# B&R Automation Studio project Parker_BMM_ST_V5_3147_V12 (part 29)

#### multsave.c
```c
/*************************************************************************************
 * COPYRIGHT --  B&R China
 *************************************************************************************
 * Program: multsave
 * File: multsave.c
 * Author: lijianjun
 * Created: March 06, 2013
 **************************************************************************************
 * Implementation of program multsave --- mold data save/load
 *************************************************************************************/

#include <bur/plctypes.h>
#include <string.h>

#ifdef _DEFAULT_INCLUDES
	#include <AsDefault.h>
#endif

#include "recipe.h"

/**************************************************************************************
** 					 	           macro define								                   **
**************************************************************************************/
#define	S$PVNAME_LENGTH		(C_PVNAME_LENGTH +1)
#define	S$LINE_NUMBER		   (C_LINE_NUMBER   +1)

#define S$WAIT_COMMAND			   10

#define S$ROOT_DISK_SAVE		   100
#define S$ROOT_DISK_LOAD		   200
#define S$ROOT_DISK_CLEAR		   500

#define S$USB_SINGLE_OPEN_SAVE	1000
#define S$USB_SINGLE_CREATE		1100
#define S$USB_SINGLE_WRITE_MEM	1200
#define S$USB_SINGLE_WRITE		   1300

#define S$USB_SINGLE_OPEN_LOAD	2000
#define S$USB_SINGLE_READ_MEM	   2100
#define S$USB_SINGLE_READ			2200

#define S$USB_SINGLE_CLOSE		   3000

#define S$USB_ALL_OPEN_SAVE	   11000
#define S$USB_ALL_CREATE		   11100
#define S$USB_ALL_MEM_ALLOC	   11200
#define S$USB_ALL_MEM_GET	      11300
#define S$USB_ALL_WRITE		      11400
#define S$USB_ALL_MEM_FREE		   11500

#define S$USB_ALL_OPEN_LOAD	   12000
#define S$USB_ALL_ALLOC_MEM	   12100
#define S$USB_ALL_READ			   12200
#define S$USB_ALL_READ_WRITE	   12300
#define S$USB_ALL_FREE_MEM  	   12400

#define S$USB_ALL_CLOSE		      13000

#define S$ERROR_STEP			      40000
/**************************************************************************************
**                            Function Declarations								     **
**************************************************************************************/
void fun_pv_name ();
void fun_pv_info ();
void fun_pv_save (unsigned short index);
void fun_pv_read (unsigned short index);
void fun_pv_clear(unsigned short index);

/**************************************************************************************
****	        		I N I T U P  O F   T H E   T A S K 		 				   ****
**************************************************************************************/
void _INIT _init(void)
{
	memset(pvList,0,sizeof(pvList));
	strcpy(pv_get.modname,"var_mold");

   strcpy(fileSingleName, "mold.usb");		/* file name */
   strcpy(fileAllName, "moldAll.usb");		/* file name */

   strcpy(DataObjOperate.ModName,"recMold");
   strcpy(DataObjOperate.Status,"");
   DataObjOperate.InitStep = 100;

   gUserPara.VarNew = 0;
}  /* end of _INIT */

/**************************************************************************************
****				C Y C L I C   P A R T   O F   T H E   T A S K  				   ****
**************************************************************************************/
void _CYCLIC _cyclic(void)
{
   pMoldUSBData = (UDINT )&tempMoldMem[0];

   /* --------------------	Step machine -- INIT -------------------- */
	switch(DataObjOperate.InitStep)
	{
		case 0:
			break;

		case 100:
			fun_pv_name ();
			if (pv_get.errorNum != 0)
			{
				DataObjOperate.InitStep = 40000;
			}
			else
			{
				DataObjOperate.InitStep = 200;
			}
			break;

		case 200:
			fun_pv_info ();
			if (pv_get.errorNum != 0)
			{
				DataObjOperate.InitStep = 40001;
			}
			else
			{
				DataObjOperate.InitStep = 300;
			}
			break;

		case 300:
         DOInfo.enable	= 1;
         DOInfo.pName	= (UDINT)DataObjOperate.ModName;
         /* Call  FUB  */
         DatObjInfo(&DOInfo);
         if (doERR_MODULNOTFOUND == DOInfo.status)	/* Data module not found -> create a new one */
         {
            DataObjOperate.InitStep  = 400;
         }
         else if (0 == DOInfo.status)
         {
            DataObjOperate.Ident = DOInfo.ident;
            DataObjOperate.InitStep = 800;
         }
         else if(DOInfo.status != ERR_FUB_BUSY)
         {
            DataObjOperate.InitStep = 40002;
         }
			break;

		case 400:
			 /* Initialize create structure */
			 DOCreate.enable 	= 1;
			 DOCreate.grp	 	= 0;
			 DOCreate.pName 	= (UDINT)DataObjOperate.ModName;
	 		 DOCreate.len 		= sizeVarSum * (S$NUM_RECIPE + 1);
			 DOCreate.MemType 	= doUSRROM;
			 DOCreate.Option 	= 0;
			 DOCreate.pCpyData 	= 0;
			 /* Call FUB */
			 DatObjCreate(&DOCreate);
			 /* Get FUB output information */
	 		 wCreate  = DOCreate.status;
	 		 if( 0 == DOCreate.status)
	 		 {
			 	DataObjOperate.Ident = DOCreate.ident;
		 	 	DataObjOperate.InitStep = 500;
		 	 }
			break;

		case 500:
			status_tmpalloc = TMP_alloc(sizeVarSum * (S$NUM_RECIPE + 1), (void*)&pData);
			if(0 == status_tmpalloc)
			{
				memset((void*)pData,0,sizeVarSum * (S$NUM_RECIPE + 1));
				DataObjOperate.InitStep = 600;
			}
			else
			{
				DataObjOperate.InitStep = 40003;
			}
			break;

		case 600:
			DOWrite.enable  = 1;
			DOWrite.ident 	 = DataObjOperate.Ident;
			DOWrite.Offset  = 0;
			DOWrite.pSource = (UDINT)pData;
			DOWrite.len 	= sizeVarSum * (S$NUM_RECIPE + 1);

			/* Call FUB */
			DatObjWrite(&DOWrite);

			if(0 == DOWrite.status)
			{
				DataObjOperate.InitStep = 700;
			}
			break;

		case 700:
			status_tmpfree = TMP_free(sizeVarSum * (S$NUM_RECIPE + 1), (void*)pData);
			if(0 == status_tmpfree)
			{
				DataObjOperate.InitStep = 800;
			}
			else
			{
				DataObjOperate.InitStep = 40004;
			}
			break;

		case 800:
			if(1 == gRecipeOperate.NameOk)
			{
				DataObjOperate.InitStep = 900;
			}
			break;

      case 900:
         fun_pv_read(S$NUM_RECIPE);
			RMold.Carriage.ValveLinear.update = 1;
			RMold.Carriage.ValveLinear.update = 1;
         gRecipeOperate.DataOk   = 1;
         DataObjOperate.InitStep = 1000;
         break;

      case 1000:
         DataObjOperate.Step = S$WAIT_COMMAND;
         DataObjOperate.InitStep = 3000;
         break;

      case 3000:
         break;
	}/* switch(DataObjOperate.InitStep) */

   if(DataObjOperate.Ident == 0 || DataObjOperate.InitStep != 3000)
   {
		gRecipeOperate.DataLoad = 0;
		gRecipeOperate.DataSave = 0;
      gRecipeOperate.DataRecipeLoad = 0;
      gRecipeOperate.DataRecipeSave = 0;
      gRecipeOperate.DataRecipeClear = 0;
      gRecipeOperate.DataUSBLoad = 0;
      gRecipeOperate.DataUSBSave = 0;
      return;
   }/* if(DataObjOperate.Ident == 0 || DataObjOperate.InitStep != 3000) */

   if(sizeVarSum > C_MEM_MOLD_LENGTH + 1)
   {
      gAlarm.RecMoldLengthErr = 1;
      return;
   }
   else
   {
      gAlarm.RecMoldLengthErr = 0;
      sizeVarSumUSB = C_MEM_MOLD_LENGTH + 1;
   }

   /* recipe save or load command  */
   switch (DataObjOperate.Step)
   {
      case S$WAIT_COMMAND:
         gRecipeOperate.usbMoldOk = 1;
         if(1 == gRecipeOperate.DataSave)
         {
            gRecipeOperate.DataSave = 0;
            indexRecipe = S$NUM_RECIPE;    	/*  current recipe in data module-index = S$NUM_RECIPE */
            DataObjOperate.Step = S$ROOT_DISK_SAVE;
         }
			else if(1 == gRecipeOperate.DataLoad)
			{
				gRecipeOperate.DataLoad = 0;
				indexRecipe = S$NUM_RECIPE;    	/*  current recipe in data module-index = S$NUM_RECIPE */
				DataObjOperate.Step = S$ROOT_DISK_LOAD;
			}
         else if(1 == gRecipeOperate.DataRecipeLoad)
         {
            gRecipeOperate.DataRecipeLoad = 0;
            indexRecipe = gRecipeOperate.Index % S$NUM_RECIPE;
            DataObjOperate.Step = S$ROOT_DISK_LOAD;
            gRecipeOperate.DataSave = 1;	/*  read from recipe then write to current recipe(S$NUM_RECIPE) in data module */
         }/* else if(1 == gRecipeOperate.DataRecipeLoad) */
         else if(1 == gRecipeOperate.DataRecipeSave)
         {
            gRecipeOperate.DataRecipeSave = 0;
            indexRecipe = gRecipeOperate.Index % S$NUM_RECIPE;
            DataObjOperate.Step = S$ROOT_DISK_SAVE;
         }/* else if(1 == gRecipeOperate.DataRecipeSave) */
         else if(1 == gRecipeOperate.DataRecipeClear)
         {
            gRecipeOperate.DataRecipeClear = 0;
            indexRecipe = gRecipeOperate.Index % S$NUM_RECIPE;
            DataObjOperate.Step = S$ROOT_DISK_CLEAR;
         }/* else if(1 == gRecipeOperate.DataLoad) */
         else if(1 == gRecipeOperate.DataUSBLoad)
         {
            gRecipeOperate.usbMoldOk = 0;
            gRecipeOperate.DataUSBLoad = 0;
            DataObjOperate.Step = S$USB_SINGLE_OPEN_LOAD;
            gRecipeOperate.DataSave = 1;	/*  read from USB then write to current recipe(S$NUM_RECIPE) in data module */
         }/* else if(1 == gRecipeOperate.DataUSBLoad) */
         else if(1 == gRecipeOperate.DataUSBSave)
         {
            gRecipeOperate.usbMoldOk = 0;
            gRecipeOperate.DataUSBSave = 0;
            DataObjOperate.Step = S$USB_SINGLE_OPEN_SAVE;
         }/* if(1 == gRecipeOperate.DataUSBSave) */
         else if(1 == gRecipeOperate.DataUSBLoadAll)
         {
            gRecipeOperate.usbMoldOk = 0;
            gRecipeOperate.DataUSBLoadAll = 0;
            DataObjOperate.Step = S$USB_ALL_OPEN_LOAD;
         }
         else if(1 == gRecipeOperate.DataUSBSaveAll)
         {
            gRecipeOperate.usbMoldOk = 0;
            gRecipeOperate.DataUSBSaveAll = 0;
            DataObjOperate.Step = S$USB_ALL_OPEN_SAVE;
         }
         break;

      /* ---------------- Save to data object ---------------- */
      case S$ROOT_DISK_SAVE:
         fun_pv_save(indexRecipe);
         DataObjOperate.Step = S$WAIT_COMMAND;
         break;

      /* ---------------- Load from data object ---------------- */
      case S$ROOT_DISK_LOAD:
         fun_pv_read (indexRecipe);
         DataObjOperate.Step = S$WAIT_COMMAND;
         break;

      /* ---------------- clear data object part ---------------- */
      case S$ROOT_DISK_CLEAR:
         fun_pv_clear(indexRecipe);
         DataObjOperate.Step = S$WAIT_COMMAND;
         break;
		/* --------------------------------------------------------- */
      /* ---------------- Single Save to usb disk ---------------- */
      /* --------------------------------------------------------- */
      case S$USB_SINGLE_OPEN_SAVE:			/* file OPEN for save  */
         FileOpen_0.enable  = 1;
         FileOpen_0.pDevice = (UDINT)&gRecipeOperate.deviceNameUSB;
         FileOpen_0.pFile   = (UDINT)&fileSingleName;
         FileOpen_0.mode    = fiREAD_WRITE;

         /* Call FUB */
         FileOpen(&FileOpen_0);

         if(fiERR_FILE_NOT_FOUND == FileOpen_0.status)/* no file   */
         {
            FileOpen_0.enable  = 0;
            DataObjOperate.Step = S$USB_SINGLE_CREATE;
         }
         else
         {
            if(ERR_OK == FileOpen_0.status)			/* file exist */
            {
               FileOpen_0.enable  = 0;
               if(FileOpen_0.filelen == sizeVarSumUSB)
               {
                  DataObjOperate.IdentUSB = FileOpen_0.ident;
                  DataObjOperate.Step = S$USB_SINGLE_WRITE_MEM;
               }
               else
               {
                  gImply.ParaUSB_Length = 1;
                  DataObjOperate.Step = S$USB_SINGLE_CLOSE;
               }
            }
            else if (FileOpen_0.status != ERR_FUB_BUSY)
            {
               FileOpen_0.enable  = 0;
               gImply.ParaOP_False = 1;
               DataObjOperate.Step = S$ERROR_STEP;
            }
         }
         break;

      case S$USB_SINGLE_CREATE:			/* file not exist, create*/
         FileCreate_0.enable  = 1;
         FileCreate_0.pDevice = (UDINT)&gRecipeOperate.deviceNameUSB;
         FileCreate_0.pFile   = (UDINT)&fileSingleName;

         /* Call FUB */
         FileCreate(&FileCreate_0);

         if(ERR_OK == FileCreate_0.status)		/* ok */
         {
            FileCreate_0.enable = 0;
            DataObjOperate.IdentUSB = FileCreate_0.ident;
            DataObjOperate.Step = S$USB_SINGLE_WRITE_MEM;
         }
         else if (FileCreate_0.status != ERR_FUB_BUSY)
         {
            FileCreate_0.enable = 0;
            gImply.ParaOP_False = 1;
            DataObjOperate.Step = S$USB_SINGLE_CLOSE;
         }
         break;

      case S$USB_SINGLE_WRITE_MEM:	/* file request single memory */
         if(pMoldUSBData != 0)
         {
            memset((void *)pMoldUSBData,0,sizeVarSumUSB);
            temp_adr_offset = 0;
            for(iLine = 0;iLine < S$LINE_NUMBER;iLine ++)
               {
               if (pv_len[iLine] != 0 && pv_adr[iLine] != 0)
               {
                  memcpy((void *)(pMoldUSBData + temp_adr_offset), (void *)pv_adr[iLine], pv_len[iLine]);
                  temp_adr_offset = temp_adr_offset + pv_len[iLine];
               }
               else break;
            }
            DataObjOperate.Step = S$USB_SINGLE_WRITE;
         }
         else
         {
            gImply.ParaOP_False = 1;
            DataObjOperate.Step = S$USB_SINGLE_CLOSE;
         }
         break;

      case S$USB_SINGLE_WRITE:		/* file single write */
         FileWrite_0.enable = 1;
         FileWrite_0.ident  = DataObjOperate.IdentUSB;
         FileWrite_0.offset = 0;
         FileWrite_0.pSrc = (UDINT)pMoldUSBData;
         FileWrite_0.len  = sizeVarSumUSB;

         /* Call FUB */
         FileWrite(&FileWrite_0);

         if(ERR_OK == FileWrite_0.status)				/* ok */
         {
            FileWrite_0.enable = 0;
            gImply.ParaOP_OK = 1;
            DataObjOperate.Step = S$USB_SINGLE_CLOSE;
         }
         else if (FileWrite_0.status != ERR_FUB_BUSY)
         {
            FileWrite_0.enable = 0;
            gImply.ParaOP_False = 1;
            DataObjOperate.Step = S$USB_SINGLE_CLOSE;
         }
         break;

      /* ----------------------------------------------------------- */
      /* ---------------- Single Load from USB disk ---------------- */
      /* ----------------------------------------------------------- */
      case S$USB_SINGLE_OPEN_LOAD:			/* file OPEN  for load  */
         FileOpen_0.enable  = 1;
         FileOpen_0.pDevice = (UDINT)&gRecipeOperate.deviceNameUSB;
         FileOpen_0.pFile   = (UDINT)&fileSingleName;
         FileOpen_0.mode    = fiREAD_WRITE;

         /* Call FUB */
         FileOpen(&FileOpen_0);

         if(fiERR_FILE_NOT_FOUND == FileOpen_0.status)	/* no file   */
         {
            FileOpen_0.enable  = 0;
            gImply.ParaUSB_NoFile = 1;
            DataObjOperate.Step = S$WAIT_COMMAND;
         }
         else
         {
            if(ERR_OK == FileOpen_0.status)				/* file exist */
            {
               FileOpen_0.enable = 0;
               if(FileOpen_0.filelen == sizeVarSumUSB)
               {
                  DataObjOperate.IdentUSB = FileOpen_0.ident;
                  DataObjOperate.Step = S$USB_SINGLE_READ_MEM;
               }
               else
               {
                  gImply.ParaUSB_Length = 1;
                  DataObjOperate.Step = S$USB_SINGLE_CLOSE;
               }
            }
            else if (FileOpen_0.status != ERR_FUB_BUSY)
            {
               FileOpen_0.enable = 0;
               gImply.ParaOP_False = 1;
               DataObjOperate.Step = S$ERROR_STEP;
            }
         }
         break;

      case S$USB_SINGLE_READ_MEM:			/* file  read request memory */
         if(pMoldUSBData != 0)
         {
            DataObjOperate.Step = S$USB_SINGLE_READ;
         }
         else
         {
            gImply.ParaOP_False = 1;
            DataObjOperate.Step = S$USB_SINGLE_CLOSE;
         }
         break;

      case S$USB_SINGLE_READ:			/* file  read  */
         FileRead_0.enable = 1;
         FileRead_0.ident  = DataObjOperate.IdentUSB;
         FileRead_0.offset = 0;
         FileRead_0.pDest  = (UDINT)pMoldUSBData;
         FileRead_0.len    = sizeVarSumUSB;

         /* Call FUB */
         FileRead(&FileRead_0);

         if(ERR_OK == FileRead_0.status)	/* ok */
         {
            FileRead_0.enable = 0;
            temp_adr_offset = 0;
            for(iLine = 0;iLine < S$LINE_NUMBER;iLine ++)
               {
               if (pv_len[iLine] != 0 && pv_adr[iLine] != 0)
               {
                  memcpy((void *)pv_adr[iLine],(void *)(pMoldUSBData + temp_adr_offset), pv_len[iLine]);
                  temp_adr_offset = temp_adr_offset + pv_len[iLine];
               }
               else break;
            }
            gImply.ParaOP_OK = 1;

				gRecipeOperate.DataSave = 1;
				gRecipeOperate.NameLoad = 1;

            /*gRecipeOperate.DataSave = 1;*/
            DataObjOperate.Step = S$USB_SINGLE_CLOSE;
         }
         else if (FileRead_0.status != ERR_FUB_BUSY)
         {
            FileRead_0.enable = 0;
            gImply.ParaOP_False = 1;
            DataObjOperate.Step = S$USB_SINGLE_CLOSE;
         }
         break;
		/* -------------------------------------------------------------- */
      /* ---------------- Single Close USB file device ---------------- */
      /* -------------------------------------------------------------- */
      case S$USB_SINGLE_CLOSE:			/* file close*/
         FileClose_0.enable = 1;
         FileClose_0.ident  = DataObjOperate.IdentUSB;

         /* Call FBK */
         FileClose(&FileClose_0);

         if(ERR_OK == FileClose_0.status)	/* ok */
         {
            FileClose_0.enable = 0;
            DataObjOperate.Step = S$WAIT_COMMAND;
         }
         else if (FileClose_0.status != ERR_FUB_BUSY)
         {
            FileClose_0.enable = 0;
            DataObjOperate.Step = S$ERROR_STEP;
         }
         break;
      /* ------------------------------------------------------ */
      /* ---------------- All Save to usb disk ---------------- */
      /* ------------------------------------------------------ */
      case S$USB_ALL_OPEN_SAVE:			/* file OPEN for save  */
         FileOpen_0.enable  = 1;
         FileOpen_0.pDevice = (UDINT)&gRecipeOperate.deviceNameUSB;
         FileOpen_0.pFile   = (UDINT)&fileAllName;
         FileOpen_0.mode    = fiREAD_WRITE;

         /* Call FUB */
         FileOpen(&FileOpen_0);

         if(fiERR_FILE_NOT_FOUND == FileOpen_0.status)/* no file   */
         {
            FileOpen_0.enable  = 0;
            DataObjOperate.Step = S$USB_ALL_CREATE;
         }
         else
         {
            if(ERR_OK == FileOpen_0.status)			/* file exist */
            {
               FileOpen_0.enable  = 0;
               if(FileOpen_0.filelen == sizeVarSum * (S$NUM_RECIPE + 1))
               {
                  DataObjOperate.IdentAllUSB = FileOpen_0.ident;
                  DataObjOperate.Step = S$USB_ALL_MEM_ALLOC;
               }
               else
               {
                  gImply.ParaUSB_Length = 1;
                  DataObjOperate.Step = S$USB_ALL_CLOSE;
               }
            }
            else if (FileOpen_0.status != ERR_FUB_BUSY)
            {
               FileOpen_0.enable  = 0;
               gImply.ParaOP_False = 1;
               DataObjOperate.Step = S$ERROR_STEP;
            }
         }
         break;

      case S$USB_ALL_CREATE:			/* file not exist, create*/
         FileCreate_0.enable  = 1;
         FileCreate_0.pDevice = (UDINT)&gRecipeOperate.deviceNameUSB;
         FileCreate_0.pFile   = (UDINT)&fileAllName;

         /* Call FUB */
         FileCreate(&FileCreate_0);

         if(ERR_OK == FileCreate_0.status)		/* ok */
         {
            FileCreate_0.enable = 0;
            DataObjOperate.IdentAllUSB = FileCreate_0.ident;
            DataObjOperate.Step = S$USB_ALL_MEM_ALLOC;
         }
         else if (FileCreate_0.status != ERR_FUB_BUSY)
         {
            FileCreate_0.enable = 0;
            gImply.ParaOP_False = 1;
            DataObjOperate.Step = S$USB_ALL_CLOSE;
         }
         break;

      case S$USB_ALL_MEM_ALLOC:	/* file request All memory */
         status_tmpalloc = TMP_alloc(sizeVarSum * (S$NUM_RECIPE + 1), (void*)&pData);
         if(0 == status_tmpalloc)
         {
            memset((void *)pData,0,sizeVarSum * (S$NUM_RECIPE + 1));
            DataObjOperate.Step = S$USB_ALL_MEM_GET;
         }
         else
         {
            gImply.ParaOP_False = 1;
            DataObjOperate.Step = S$USB_ALL_CLOSE;
         }
         break;

      case S$USB_ALL_MEM_GET:
         DORead.enable = 1;
         DORead.ident  = DataObjOperate.Ident;
         DORead.Offset = 0;
         DORead.pDestination = (UDINT)pData;
         DORead.len = sizeVarSum * (S$NUM_RECIPE + 1);

         /* Call FUB */
         DatObjRead(&DORead);
         if(0 == DORead.status)
         {
            DORead.enable = 0;
            DataObjOperate.Step = S$USB_ALL_WRITE;
         }
         else if (DORead.status != ERR_FUB_BUSY)
         {
            DORead.enable = 0;
            gImply.ParaOP_False = 1;
            DataObjOperate.Step = S$USB_ALL_MEM_FREE;
         }
         break;

      case S$USB_ALL_WRITE:		/* file single write */
         FileWrite_0.enable = 1;
         FileWrite_0.ident  = DataObjOperate.IdentAllUSB;
         FileWrite_0.offset = 0;
         FileWrite_0.pSrc = (UDINT)pData;
         FileWrite_0.len  = sizeVarSum * (S$NUM_RECIPE + 1);

         /* Call FUB */
         FileWrite(&FileWrite_0);

         if(ERR_OK == FileWrite_0.status)				/* ok */
         {
            FileWrite_0.enable = 0;
            gImply.ParaOP_OK = 1;
            DataObjOperate.Step = S$USB_ALL_MEM_FREE;
         }
         else if (FileWrite_0.status != ERR_FUB_BUSY)
         {
            FileWrite_0.enable = 0;
            gImply.ParaOP_False = 1;
            DataObjOperate.Step = S$USB_ALL_MEM_FREE;
         }
         break;

      case S$USB_ALL_MEM_FREE:
         status_tmpfree = TMP_free(sizeVarSum * (S$NUM_RECIPE + 1), (void*)pData);
         if(0 == status_tmpfree)
         {
            DataObjOperate.Step = S$USB_ALL_CLOSE;
         }
         else
         {
            DataObjOperate.Step = S$USB_ALL_CLOSE;
         }
         break;

      /* ----------------------------------------------------------- */
      /* ----------------  All Load from USB disk   ---------------- */
      /* ----------------------------------------------------------- */
      case S$USB_ALL_OPEN_LOAD:			/* file OPEN  for load  */
         FileOpen_0.enable  = 1;
         FileOpen_0.pDevice = (UDINT)&gRecipeOperate.deviceNameUSB;
         FileOpen_0.pFile   = (UDINT)&fileAllName;
         FileOpen_0.mode    = fiREAD_WRITE;

         /* Call FUB */
         FileOpen(&FileOpen_0);

         if(fiERR_FILE_NOT_FOUND == FileOpen_0.status)	/* no file   */
         {
            FileOpen_0.enable  = 0;
            gImply.ParaUSB_NoFile = 1;
            DataObjOperate.Step = S$WAIT_COMMAND;
         }
         else
         {
            if(ERR_OK == FileOpen_0.status)				/* file exist */
            {
               FileOpen_0.enable = 0;
               if(FileOpen_0.filelen == sizeVarSum * (S$NUM_RECIPE + 1))
               {
                  DataObjOperate.IdentAllUSB = FileOpen_0.ident;
                  DataObjOperate.Step = S$USB_ALL_ALLOC_MEM;
               }
               else
               {
                  gImply.ParaUSB_Length = 1;
                  DataObjOperate.Step = S$USB_ALL_CLOSE;
               }
            }
            else if (FileOpen_0.status != ERR_FUB_BUSY)
            {
               FileOpen_0.enable = 0;
               gImply.ParaOP_False = 1;
               DataObjOperate.Step = S$ERROR_STEP;
            }
         }
         break;

      case S$USB_ALL_ALLOC_MEM:			/* file  read request memory */
         status_tmpalloc = TMP_alloc(sizeVarSum * (S$NUM_RECIPE + 1), (void*)&pData);
         if(0 == status_tmpalloc)
         {
            DataObjOperate.Step = S$USB_ALL_READ;
         }
         else
         {
            gImply.ParaOP_False = 1;
            DataObjOperate.Step = S$USB_ALL_CLOSE;
         }
         break;

      case S$USB_ALL_READ:			/* file  read  */
         FileRead_0.enable = 1;
         FileRead_0.ident  = DataObjOperate.IdentAllUSB;
         FileRead_0.offset = 0;
         FileRead_0.pDest  = (UDINT)pData;
         FileRead_0.len    = sizeVarSum * (S$NUM_RECIPE + 1);

         /* Call FUB */
         FileRead(&FileRead_0);

         if(ERR_OK == FileRead_0.status)	/* ok */
         {
            FileRead_0.enable = 0;
            DataObjOperate.Step = S$USB_ALL_READ_WRITE;
         }
         else if (FileRead_0.status != ERR_FUB_BUSY)
         {
            FileRead_0.enable = 0;
            gImply.ParaOP_False = 1;
            DataObjOperate.Step = S$USB_ALL_FREE_MEM;
         }
         break;

      case S$USB_ALL_READ_WRITE:
         DOWrite.enable  = 1;
         DOWrite.ident 	 = DataObjOperate.Ident;
         DOWrite.Offset  = 0;
         DOWrite.pSource = (UDINT)pData;
         DOWrite.len 	= sizeVarSum * (S$NUM_RECIPE + 1);

         DatObjWrite(&DOWrite);

         if(0 == DOWrite.status)
         {
            DOWrite.enable  = 0;
            gImply.ParaOP_OK = 1;
				gRecipeOperate.DataLoad = 1;
            DataObjOperate.Step = S$USB_ALL_FREE_MEM;
         }
         else if (DOWrite.status != ERR_FUB_BUSY)
         {
            DOWrite.enable  = 0;
            gImply.ParaOP_False = 1;
            DataObjOperate.Step = S$USB_ALL_FREE_MEM;
         }
         break;

      case S$USB_ALL_FREE_MEM:
         status_tmpfree = TMP_free(sizeVarSum * (S$NUM_RECIPE + 1), (void*)pData);
         if(0 == status_tmpfree)
         {
            DataObjOperate.Step = S$USB_ALL_CLOSE;
         }
         else
         {
            DataObjOperate.Step = S$USB_ALL_CLOSE;
         }
         break;
		/* ----------------------------------------------------------- */
      /* ---------------- All Close USB file device ---------------- */
      /* ----------------------------------------------------------- */
      case S$USB_ALL_CLOSE:			/* file close*/
         FileClose_0.enable = 1;
         FileClose_0.ident  = DataObjOperate.IdentAllUSB;

         /* Call FBK */
         FileClose(&FileClose_0);

         if(ERR_OK == FileClose_0.status)	/* ok */
         {
            FileClose_0.enable = 0;
            DataObjOperate.Step = S$WAIT_COMMAND;
         }
         else if (FileClose_0.status != ERR_FUB_BUSY)
         {
            FileClose_0.enable = 0;
            DataObjOperate.Step = S$ERROR_STEP;
         }
         break;

      case S$ERROR_STEP:
            DataObjOperate.Step = S$WAIT_COMMAND;
         break;
   }/* switch (DataObjOperate.Step) */

}  /* end of _CYCLIC */

void fun_pv_name ()
{
   DOInfo.enable	= 1;
   DOInfo.pName 	= (UDINT)pv_get.modname;
   DatObjInfo(&DOInfo);

   if (DOInfo.status!= 0)
   {
      pv_get.errorNum = 1000; /*can not find the config data*/
      return;
   }

   while (iLine < DOInfo.len/S$PVNAME_LENGTH)
   {
      strcpy(pvList[iLine],(char*)(DOInfo.pDatObjMem+iLine*S$PVNAME_LENGTH));
         iLine++;
   }
}/* end of function */

void fun_pv_info ()
{
   sizeVarSum = 0;
   memset(pv_adr,0,sizeof(pv_adr));
   memset(pv_len,0,sizeof(pv_len));

   for (iLine = 0;iLine < DOInfo.len/S$PVNAME_LENGTH;iLine++)
   {
      status = PV_xgetadr(pvList[iLine], &pv_adr[iLine], &pv_len[iLine]);
      if (status == 0)
      {
         sizeVarSum = sizeVarSum + pv_len[iLine];
      }
      else if (status == 14700) /*Invalid PV name*/
      {
         if(sizeVarSum < C_MEM_MOLD_LENGTH - 191)
         {
            sizeVarSum = C_MEM_MOLD_LENGTH - 191;
         }
         else
         {
            pv_get.errorNum = 2001;
         }
         break;
      }
      else if (status != 0)
      {
         pv_get.errorNum = 2000;
         pv_get.line_no  = iLine + 1;
         return;
      }
   }
}/* end of _function */

void fun_pv_save (unsigned short index)
{
   status = TMP_alloc(sizeVarSum, (void*)&(temp_adr));

   if (status != 0) return;

   temp_adr_offset = 0;

   for(iLine = 0;iLine < S$LINE_NUMBER;iLine ++)
      {
      if (pv_len[iLine] != 0 && pv_adr[iLine] != 0)
      {
         memcpy((void *)(temp_adr + temp_adr_offset), (void *)pv_adr[iLine], pv_len[iLine]);
         temp_adr_offset = temp_adr_offset + pv_len[iLine];
      }
      else break;
   }

   /* Initialize write structure */
   DOWrite.enable 	= 1;
   DOWrite.ident 	    = DataObjOperate.Ident;
   DOWrite.Offset 	= sizeVarSum*index;
   DOWrite.pSource    = (UDINT)temp_adr;
   DOWrite.len 	    = sizeVarSum;
   DatObjWrite(&DOWrite);
   wWrite = DOWrite.status;

   status = TMP_free(sizeVarSum, (void*)temp_adr);

}/* end of _function */

void fun_pv_read (unsigned short index)
{
   status = TMP_alloc(sizeVarSum, (void*)&(temp_adr));

   if (status != 0) return;

   temp_adr_offset = 0;

   /* Initialize read structure */
   DORead.enable 		= 1;
   DORead.ident 		= DataObjOperate.Ident;
   DORead.Offset 		= sizeVarSum*index;
   DORead.pDestination	= (UDINT)temp_adr;
   DORead.len 			= sizeVarSum;

   /* Call FUB */
   DatObjRead(&DORead);

   /* Get status */
   wRead = DORead.status;

   for(iLine = 0;iLine < S$LINE_NUMBER;iLine ++)
      {
      if (pv_len[iLine] != 0 && pv_adr[iLine] != 0)
      {
         memcpy((void *)pv_adr[iLine],(void *)(temp_adr + temp_adr_offset), pv_len[iLine]);
         temp_adr_offset = temp_adr_offset + pv_len[iLine];
      }
      else break;
   }

   status = TMP_free(sizeVarSum, (void*)temp_adr);

}/* end of _function */

void fun_pv_clear (unsigned short index)
{
   status = TMP_alloc(sizeVarSum, (void*)&(temp_adr));

   if (status != 0) return;

   memset((void *)temp_adr,0,sizeVarSum);

   /* Initialize write structure */
   DOWrite.enable 	= 1;
   DOWrite.ident 	    = DataObjOperate.Ident;
   DOWrite.Offset 	= sizeVarSum*index;
   DOWrite.pSource    = (UDINT)temp_adr;
   DOWrite.len 	    = sizeVarSum;
   DatObjWrite(&DOWrite);
   wWrite = DOWrite.status;

   status = TMP_free(sizeVarSum, (void*)temp_adr);

}/* void fun_pv_clear (unsigned short index) */
```

#### multsave.var
```iecst
VAR
	DataObjOperate : DatObj_Operate_typ;
	indexRecipe : UINT;
	pData : UDINT;
	status_tmpalloc : UINT;
	status_tmpfree : UINT;
	pv_get : pv_get_typ;
	pvList : ARRAY[0..C_LINE_NUMBER] OF STRING[C_PVNAME_LENGTH];
	pv_adr : ARRAY[0..C_LINE_NUMBER] OF UDINT;
	pv_len : ARRAY[0..C_LINE_NUMBER] OF UDINT;
	iLine : UINT;
	status : UINT;
	wCreate : UINT;
	wWrite : UINT;
	wRead : UINT;
	DOCreate : DatObjCreate;
	DOWrite : DatObjWrite;
	DORead : DatObjRead;
	DOInfo : DatObjInfo;
	sizeVarSum : UDINT;
	sizeVarSumUSB : UDINT;
	temp_adr : UDINT;
	temp_adr_offset : UDINT;
	pMoldUSBData : UDINT;
	fileSingleName : STRING[80];
	fileAllName : STRING[80];
	FileCreate_0 : FileCreate;
	FileWrite_0 : FileWrite;
	FileRead_0 : FileRead;
	FileOpen_0 : FileOpen;
	FileClose_0 : FileClose;
	tempMoldMem : ARRAY[0..C_MEM_MOLD_LENGTH] OF UINT;
END_VAR
```

### Program Logical/recipeMan/oncesave (ANSIC, version 1.00.0) - fix dada load/save

#### oncesave.c
```c
/***************************************************************************************
 * COPYRIGHT --  B&R China
 **************************************************************************************
 * Program: oncesave
 * File: oncesave.c
 * Author: lijianjun
 * Created: March 06, 2013
 **************************************************************************************
 * Implementation of program oncesave --- Fix data load/save
 *************************************************************************************/

#include <bur/plctypes.h>
#include <string.h>

#ifdef _DEFAULT_INCLUDES
	#include <AsDefault.h>
#endif

#include "recipe.h"

/**************************************************************************************
** 					 	          macro define								                   **
**************************************************************************************/
#define	S$PVNAME_LENGTH		(C_PVNAME_LENGTH + 1)
#define	S$LINE_NUMBER		   (C_LINE_NUMBER   + 1)

#define S$WAIT_COMMAND			   10

#define S$ROOT_DISK_SAVE		   100
#define S$ROOT_DISK_LOAD		   200
#define S$ROOT_DISK_CLEAR		   500

#define S$USB_SINGLE_OPEN_SAVE	1000
#define S$USB_SINGLE_CREATE		1100
#define S$USB_SINGLE_WRITE_MEM	1200
#define S$USB_SINGLE_WRITE		   1300

#define S$USB_SINGLE_OPEN_LOAD	2000
#define S$USB_SINGLE_READ_MEM	   2100
#define S$USB_SINGLE_READ			2200

#define S$USB_SINGLE_CLOSE		   3000

#define S$ERROR_STEP			      40000
/**************************************************************************************
**                            Function Declarations								          **
**************************************************************************************/
void fun_pv_name ();
void fun_pv_info ();
void fun_pv_save ();
void fun_pv_read ();
void fun_pv_clear();
/**************************************************************************************
****	        		    I N I T U P  O F   T H E   T A S K 		 				        ****
**************************************************************************************/
void _INIT _init(void)
{
   memset(pvList,0,sizeof(pvList));
   strcpy(pv_get.modname,"var_fix");
   strcpy(fileSingleName, "fix.usb");		/* file name */

   strcpy(DataObjOperate.ModName,"recFix");
   strcpy(DataObjOperate.Status,"");
   DataObjOperate.InitStep = 100;

   gUserFix.VarNew = 0;
}  /* end of _INIT */

/**************************************************************************************
****				C Y C L I C   P A R T   O F   T H E   T A S K  				           ****
**************************************************************************************/
void _CYCLIC _cyclic(void)
{
   pFixUSBData = (UDINT )&tempOnceMem[0];

   /* --------------------	Step machine -- INIT -------------------- */
	switch(DataObjOperate.InitStep)
	{
		case 0:
			break;

		case 100:
			fun_pv_name ();
			if (pv_get.errorNum != 0)
			{
				DataObjOperate.InitStep = 40000;
			}
			else
			{
				DataObjOperate.InitStep = 200;
			}
			break;

		case 200:
			fun_pv_info ();
			if (pv_get.errorNum != 0)
			{
				DataObjOperate.InitStep = 40001;
			}
			else
			{
				DataObjOperate.InitStep = 300;
			}
			break;

		case 300:
			 DOInfo.enable	= 1;
			 DOInfo.pName	= (UDINT)DataObjOperate.ModName;
			 /* Call  FUB  */
			 DatObjInfo(&DOInfo);
			 if (DOInfo.status == doERR_MODULNOTFOUND)	/* Data module not found -> create a new one */
			 {
			 	 DataObjOperate.InitStep  = 400;
		 	 }
			 else
			 {
				 DataObjOperate.Ident  = DOInfo.ident;
				 DataObjOperate.InitStep = 800;
			 }
			break;

		case 400:
			 /* Initialize create structure */
			 DOCreate.enable 	= 1;
			 DOCreate.grp	 	= 0;
			 DOCreate.pName 	= (UDINT)DataObjOperate.ModName;
	 		 DOCreate.len 		= sizeVarSumFix;
			 DOCreate.MemType = doUSRROM;
			 DOCreate.Option 	= 0;
			 DOCreate.pCpyData= 0;
			 /* Call FUB */
			 DatObjCreate(&DOCreate);
			 /* Get FUB output information */
			 wCreate  = DOCreate.status;
			 if( 0 == DOCreate.status)
			 {
			 	DataObjOperate.Ident  = DOCreate.ident;
		 	 	DataObjOperate.InitStep = 500;
		 	 }
			break;

		case 500:
			status_tmpalloc = TMP_alloc(sizeVarSumFix, (void*)&pData);
			if(0 == status_tmpalloc)
			{
				memset((void*)pData,0,sizeVarSumFix);
				DataObjOperate.InitStep = 600;
			}
			else
			{
				DataObjOperate.InitStep = 40002;
			}
			break;

		case 600:
			DOWrite.enable  = 1;
			DOWrite.ident 	 = DataObjOperate.Ident;
			DOWrite.Offset  = 0;
			DOWrite.pSource = (UDINT)pData;
			DOWrite.len 	= sizeVarSumFix;

			/* Call FUB */
			DatObjWrite(&DOWrite);

			if(0 == DOWrite.status)
			{
				DataObjOperate.InitStep = 700;
			}
			break;

		case 700:
			status_tmpfree = TMP_free(sizeVarSumFix, (void*)pData);
			if(0 == status_tmpfree)
			{
				DataObjOperate.InitStep = 800;
			}
			else
			{
				DataObjOperate.InitStep = 40003;
			}
			break;

		case 800:
			DataObjOperate.InitStep = 900;
			break;

		case 900:
			 fun_pv_read ();
			 gRecipeOperate.OnceOk = 1;
			 DataObjOperate.InitStep = 1000;
			break;

		case 1000:
         DataObjOperate.Step = S$WAIT_COMMAND;
         DataObjOperate.InitStep  = 3000;
			break;

      case 3000:
         break;

		case 9999:
			break;
	}/* switch(DataObjOperate.InitStep) */

   if(DataObjOperate.Ident == 0 || DataObjOperate.InitStep != 3000)
   {
      gRecipeOperate.OnceUSBSave = 0;
      gRecipeOperate.OnceUSBLoad = 0;
      return;
   }/* if(DataObjOperate.Ident == 0 || DataObjOperate.InitStep != 3000) */

   if(sizeVarSumFix > C_MEM_FIX_LENGTH + 1)
   {
      gAlarm.RecFixLengthErr = 1;
      return;
   }
   else
   {
      gAlarm.RecFixLengthErr = 0;
      sizeVarSumUSB = C_MEM_FIX_LENGTH + 1;
   }

   /* ----------------- Step machine control ----------------- */
   switch (DataObjOperate.Step)
   {
      case S$WAIT_COMMAND:
         gRecipeOperate.usbFixOk = 1;
         if(1 == gRecipeOperate.OnceSave)
         {
            gRecipeOperate.OnceSave = 0;
            DataObjOperate.Step = S$ROOT_DISK_SAVE;
         }/* else if(1 == gRecipeOperate.OnceSave) */
         else if(1 == gRecipeOperate.OnceLoad)
         {
            gRecipeOperate.OnceLoad = 0;
            DataObjOperate.Step = S$ROOT_DISK_LOAD;
         }/* else if(1 == gImply.OnceLoad) */
         else if(1 == gRecipeOperate.OnceUSBSave)
         {
            gRecipeOperate.usbFixOk = 0;
            gRecipeOperate.OnceUSBSave = 0;
            DataObjOperate.Step = S$USB_SINGLE_OPEN_SAVE;
         }/* else if(1 == gImply.DataUSBSave) */
         else if(1 == gRecipeOperate.OnceUSBLoad)
         {
            gRecipeOperate.usbFixOk = 0;
            gRecipeOperate.OnceUSBLoad = 0;
            DataObjOperate.Step = S$USB_SINGLE_OPEN_LOAD;
				gRecipeOperate.OnceSave = 1;
         }/* else if(1 == gImply.DataUSBLoad) */
         break;

      /* ---------------- Save to root disk ---------------- */
      case S$ROOT_DISK_SAVE:
         fun_pv_save();
         DataObjOperate.Step = S$WAIT_COMMAND;
         break;

      /* ---------------- Load from root disk ---------------- */
      case S$ROOT_DISK_LOAD:
         fun_pv_read();
         DataObjOperate.Step = S$WAIT_COMMAND;
         break;

      /* -------------------------------------------------- */
      /* ---------------- Save to usb disk ---------------- */
      /* -------------------------------------------------- */
      case S$USB_SINGLE_OPEN_SAVE:			/* file OPEN for save  */
         FileOpen_0.enable  = 1;
         FileOpen_0.pDevice = (UDINT)&gRecipeOperate.deviceNameUSB;
         FileOpen_0.pFile   = (UDINT)&fileSingleName;
         FileOpen_0.mode    = fiREAD_WRITE;

         /* Call FUB */
         FileOpen(&FileOpen_0);

         if(fiERR_FILE_NOT_FOUND == FileOpen_0.status)/* no file   */
         {
            FileOpen_0.enable  = 0;
            DataObjOperate.Step = S$USB_SINGLE_CREATE;
         }
         else
         {
            if(ERR_OK == FileOpen_0.status)			/* file exist */
            {
               FileOpen_0.enable  = 0;
               if(FileOpen_0.filelen == sizeVarSumUSB)
               {
                  DataObjOperate.IdentUSB = FileOpen_0.ident;
                  DataObjOperate.Step = S$USB_SINGLE_WRITE_MEM;
               }
               else
               {
                  gImply.FixUSB_Length = 1;
                  DataObjOperate.Step = S$USB_SINGLE_CLOSE;
               }
            }
            else if (FileOpen_0.status != ERR_FUB_BUSY)
            {
               FileOpen_0.enable  = 0;
               gImply.FixOP_False = 1;
               DataObjOperate.Step = S$ERROR_STEP;
            }
         }
         break;

      case S$USB_SINGLE_CREATE:			/* file not exist, create*/
         FileCreate_0.enable  = 1;
         FileCreate_0.pDevice = (UDINT)&gRecipeOperate.deviceNameUSB;
         FileCreate_0.pFile   = (UDINT)&fileSingleName;

         /* Call FUB */
         FileCreate(&FileCreate_0);

         if(ERR_OK == FileCreate_0.status)		/* ok */
         {
            FileCreate_0.enable = 0;
            DataObjOperate.IdentUSB = FileCreate_0.ident;
            DataObjOperate.Step = S$USB_SINGLE_WRITE_MEM;
         }
         else if (FileCreate_0.status != ERR_FUB_BUSY)
         {
            FileCreate_0.enable= 0;
            gImply.FixOP_False = 1;
            DataObjOperate.Step = S$USB_SINGLE_CLOSE;
         }
         break;

      case S$USB_SINGLE_WRITE_MEM:	/* file write request memory */
         if(pFixUSBData != 0)
         {
            temp_adr_offset = 0;
            for(iLine = 0;iLine < S$LINE_NUMBER;iLine ++)
               {
               if (pv_len[iLine] != 0 && pv_adr[iLine] != 0)
               {
                  memcpy((void *)(pFixUSBData + temp_adr_offset), (void *)pv_adr[iLine], pv_len[iLine]);
                  temp_adr_offset = temp_adr_offset + pv_len[iLine];
               }
               else break;
            }
            DataObjOperate.Step = S$USB_SINGLE_WRITE;
         }
         else
         {
            gImply.FixOP_False = 1;
            DataObjOperate.Step = S$USB_SINGLE_CLOSE;
         }
         break;

      case S$USB_SINGLE_WRITE:		/* file write */
         FileWrite_0.enable = 1;
         FileWrite_0.ident  = DataObjOperate.IdentUSB;
         FileWrite_0.offset = 0;
         FileWrite_0.pSrc = (UDINT)pFixUSBData;
         FileWrite_0.len  = sizeVarSumUSB;

         /* Call FUB */
         FileWrite(&FileWrite_0);

         if(ERR_OK == FileWrite_0.status)				/* ok */
         {
            FileWrite_0.enable = 0;
            gImply.FixOP_OK = 1;
            DataObjOperate.Step = S$USB_SINGLE_CLOSE;
         }
         else if (FileWrite_0.status != ERR_FUB_BUSY)
         {
            FileWrite_0.enable = 0;
            gImply.FixOP_False = 1;
            DataObjOperate.Step = S$USB_SINGLE_CLOSE;
         }
         break;

      /* ---------------------------------------------------- */
      /* ---------------- Load from USB disk ---------------- */
      /* ---------------------------------------------------- */
      case S$USB_SINGLE_OPEN_LOAD:			/* file OPEN  for load  */
         FileOpen_0.enable  = 1;
         FileOpen_0.pDevice = (UDINT)&gRecipeOperate.deviceNameUSB;
         FileOpen_0.pFile   = (UDINT)&fileSingleName;
         FileOpen_0.mode    = fiREAD_WRITE;

         /* Call FUB */
         FileOpen(&FileOpen_0);

         if(fiERR_FILE_NOT_FOUND == FileOpen_0.status)	/* no file   */
         {
            FileOpen_0.enable  = 0;
            gImply.FixUSB_NoFile = 1;
            DataObjOperate.Step = S$WAIT_COMMAND;
         }
         else
         {
            if(ERR_OK == FileOpen_0.status)				/* file exist */
            {
               FileOpen_0.enable = 0;
               if(FileOpen_0.filelen == sizeVarSumUSB)
               {
                  DataObjOperate.IdentUSB = FileOpen_0.ident;
                  DataObjOperate.Step = S$USB_SINGLE_READ_MEM;
               }
               else
               {
                  gImply.FixUSB_Length = 1;
                  DataObjOperate.Step = S$USB_SINGLE_CLOSE;
               }
            }
            else if (FileOpen_0.status != ERR_FUB_BUSY)
            {
               FileOpen_0.enable = 0;
               gImply.FixOP_False = 1;
               DataObjOperate.Step = S$ERROR_STEP;
            }
         }
         break;

      case S$USB_SINGLE_READ_MEM:			/* file  read request memory */
         if(0 == status_tmpalloc)
         {
            DataObjOperate.Step = S$USB_SINGLE_READ;
         }
         else
         {
            gImply.FixOP_False = 1;
            DataObjOperate.Step = S$USB_SINGLE_CLOSE;
         }
         break;

      case S$USB_SINGLE_READ:			/* file single read  */
         FileRead_0.enable = 1;
         FileRead_0.ident  = DataObjOperate.IdentUSB;
         FileRead_0.offset = 0;
         FileRead_0.pDest  = (UDINT)pFixUSBData;
         FileRead_0.len    = sizeVarSumUSB;

         /* Call FUB */
         FileRead(&FileRead_0);

         if(ERR_OK == FileRead_0.status)	/* ok */
         {
            FileRead_0.enable = 0;
            temp_adr_offset = 0;
            for(iLine = 0;iLine < S$LINE_NUMBER;iLine ++)
               {
               if (pv_len[iLine] != 0 && pv_adr[iLine] != 0)
               {
                  memcpy((void *)pv_adr[iLine],(void *)(pFixUSBData + temp_adr_offset), pv_len[iLine]);
                  temp_adr_offset = temp_adr_offset + pv_len[iLine];
               }
               else break;
            }
            gImply.FixOP_OK = 1;
            DataObjOperate.Step = S$USB_SINGLE_CLOSE;
         }
         else if (FileRead_0.status != ERR_FUB_BUSY)
         {
            FileRead_0.enable = 0;
            gImply.FixOP_False = 1;
            DataObjOperate.Step = S$USB_SINGLE_CLOSE;
         }
         break;
		/* ------------------------------------------------------- */
      /* ---------------- Close USB file device ---------------- */
      /* ------------------------------------------------------- */
      case S$USB_SINGLE_CLOSE:			/* file close*/
         FileClose_0.enable = 1;
         FileClose_0.ident  = DataObjOperate.IdentUSB;

         /* Call FBK */
         FileClose(&FileClose_0);

         if(ERR_OK == FileClose_0.status)	/* ok */
         {
            FileClose_0.enable = 0;
            DataObjOperate.Step = S$WAIT_COMMAND;
         }
         else if (FileClose_0.status != ERR_FUB_BUSY)
         {
            FileClose_0.enable = 0;
            DataObjOperate.Step = S$ERROR_STEP;
         }
         break;

      case S$ERROR_STEP:
         DataObjOperate.Step = S$WAIT_COMMAND;
         break;

   }/* switch (DataObjOperate.Step) */

}  /* end of _CYCLIC */

void fun_pv_name ()
{
   DOInfo.enable	= 1;
   DOInfo.pName 	= (UDINT)pv_get.modname;
   DatObjInfo(&DOInfo);

   if (DOInfo.status!= 0)
   {
      pv_get.errorNum = 1000; /*can not find the config data*/
      return;
   }

   while (iLine < DOInfo.len/S$PVNAME_LENGTH)
   {
      strcpy(pvList[iLine],(char*)(DOInfo.pDatObjMem+iLine*S$PVNAME_LENGTH));
      iLine++;
   }
}/* end of function */

void fun_pv_info ()
{
   sizeVarSumFix = 0;
   memset(pv_adr,0,sizeof(pv_adr));
   memset(pv_len,0,sizeof(pv_len));

   for (iLine = 0;iLine < DOInfo.len/S$PVNAME_LENGTH;iLine++)
   {
      status = PV_xgetadr(pvList[iLine], &pv_adr[iLine], &pv_len[iLine]);
      if (status == 0)
      {
         sizeVarSumFix = sizeVarSumFix + pv_len[iLine];
      }
      else if (status == 14700) /*Invalid PV name*/
      {
         if(sizeVarSumFix < C_MEM_FIX_LENGTH - 191)
         {
            sizeVarSumFix = C_MEM_FIX_LENGTH - 191;
         }
         else
         {
            pv_get.errorNum = 2001;
         }
         break;
      }
      else if (status != 0)
      {
         pv_get.errorNum = 2000;
         pv_get.line_no  = iLine + 1;
         return;
      }
   }
}/* end of _CYCLIC */

void fun_pv_read ()
{
	 status = TMP_alloc(sizeVarSumFix, (void*)&(temp_adr));

	 if (status != 0) return;

	 temp_adr_offset = 0;

	 /* Initialize read structure */
		DORead.enable 		= 1;
		DORead.ident 		= DataObjOperate.Ident;
		DORead.Offset 		= 0;
		DORead.pDestination	= (UDINT)temp_adr;
		DORead.len 			= sizeVarSumFix;

		/* Call FUB */
		DatObjRead(&DORead);

		/* Get status */
		wRead = DORead.status;

	 for(iLine = 0;iLine < S$LINE_NUMBER;iLine ++)
	 {
	 	if (pv_len[iLine] != 0 && pv_adr[iLine] != 0)
	 	{
		 	memcpy((void *)pv_adr[iLine],(void *)(temp_adr + temp_adr_offset), pv_len[iLine]);
		 	temp_adr_offset = temp_adr_offset + pv_len[iLine];
		}
		else break;
	 }

	 status = TMP_free(sizeVarSumFix, (void*)temp_adr);
}

void fun_pv_save ()
{
	 status = TMP_alloc(sizeVarSumFix, (void*)&(temp_adr));

	 if (status != 0) return;

	 temp_adr_offset = 0;

	 for(iLine = 0;iLine < S$LINE_NUMBER;iLine ++)
	 {
	 	if (pv_len[iLine] != 0 && pv_adr[iLine] != 0)
	 	{
		 	memcpy((void *)(temp_adr + temp_adr_offset), (void *)pv_adr[iLine], pv_len[iLine]);
		 	temp_adr_offset = temp_adr_offset + pv_len[iLine];
		}
		else break;
	 }

	 /* Initialize write structure */
	 DOWrite.enable 	= 1;
	 DOWrite.ident 	= DataObjOperate.Ident;
	 DOWrite.Offset 	= 0;
	 DOWrite.pSource  = (UDINT)temp_adr;
	 DOWrite.len 	   = sizeVarSumFix;
	 DatObjWrite(&DOWrite);
	 wWrite = DOWrite.status;

     status = TMP_free(sizeVarSumFix, (void*)temp_adr);
}/* end of _CYCLIC */

void fun_pv_clear ()
{
   status = TMP_alloc(sizeVarSumFix, (void*)&(temp_adr));

   if (status != 0) return;

   memset((void *)temp_adr,0,sizeVarSumFix);

   /* Initialize write structure */
   DOWrite.enable  = 1;
   DOWrite.ident 	 = DataObjOperate.Ident;
   DOWrite.Offset  = 0;
   DOWrite.pSource = (UDINT)temp_adr;
   DOWrite.len 	 = sizeVarSumFix;
   DatObjWrite(&DOWrite);
   wWrite = DOWrite.status;

   status = TMP_free(sizeVarSumFix, (void*)temp_adr);
}/* void fun_pv_clear (unsigned short index) */
```

#### oncesave.var
```iecst
VAR
	DataObjOperate : DatObj_Operate_typ;
	DOCreate : DatObjCreate;
	DOInfo : DatObjInfo;
	DORead : DatObjRead;
	DOWrite : DatObjWrite;
	pv_get : pv_get_typ;
	pvList : ARRAY[0..C_LINE_NUMBER] OF STRING[C_PVNAME_LENGTH];
	temp_adr_offset : UDINT;
	pData : UDINT;
	sizeVarSumUSB : UDINT;
	sizeVarSumFix : UDINT;
	temp_adr : UDINT;
	pv_adr : ARRAY[0..C_LINE_NUMBER] OF UDINT;
	pv_len : ARRAY[0..C_LINE_NUMBER] OF UDINT;
	wWrite : UINT;
	wRead : UINT;
	wCreate : UINT;
	status_tmpfree : UINT;
	status : UINT;
	status_tmpalloc : UINT;
	iLine : UINT;
	pFixUSBData : UDINT;
	fileSingleName : STRING[80];
	FileOpen_0 : FileOpen;
	FileCreate_0 : FileCreate;
	FileWrite_0 : FileWrite;
	FileRead_0 : FileRead;
	FileClose_0 : FileClose;
	tempOnceMem : ARRAY[0..C_MEM_FIX_LENGTH] OF USINT;
END_VAR
```

### Program Logical/recipeMan/cfg_cpy (ANSIC, version 1.00.0) - temperature default parameter load

#### cfg_cpy.typ - Local data types
```iecst
(********************************************************************
 * COPYRIGHT --  B&R CHINA
 ********************************************************************
 * Program: cfg_cpy
 * File: cfg_cpy.typ
 * Author: lij
 * Created: March 06, 2013
 ********************************************************************
 * Local data types of program cfg_cpy  --- configure parameter copy
 ********************************************************************)

TYPE
	var_rd_typ : 	STRUCT
		modname : STRING[20];
		taskname : STRING[20];
		pre_string : STRING[10];
		error : UINT;
		line_no : UINT;
		PV_name : ARRAY[0..49]OF SINT;
	END_STRUCT;
END_TYPE
```

#### cfg_cpy.c - default configure parameter copy to PLC
```c
/********************************************************************
 * COPYRIGHT --  B&R
 ********************************************************************
 * Program: cfg_cpy
 * File: cfg_cpy.c
 * Author: lijianjun
 * Created: March 06, 2013
 ********************************************************************
 * Implementation of program cfg_cpy --- copy default value to data
 ********************************************************************/

#include <bur/plctypes.h>

#ifdef _DEFAULT_INCLUDES
	#include <AsDefault.h>
#endif

#include <string.h>

#include "edge.h"

/********************************************************************
 *                                                         Function		 								                          *
********************************************************************/

unsigned short	var_rd(var_rd_typ	*var_rd_ptr);

/********************************************************************
****	       I N I T U P  O F   T H E   T A S K 		 		 ****
********************************************************************/
void _INIT Rec_cpy_init(void)
{
	wCfgLoad =1;
}  /* end of _INIT */
/********************************************************************
****	  C Y C L I C   P A R T   O F   T H E   T A S K  		 ****
********************************************************************/
void _CYCLIC Rec_cpy_cyclic(void)
{

	/*set config load command bit, for loading*/
	if (gT_Par.Fix.AT_MAX == 0 && wCfgLoad ==0) wCfgLoad =1;

	if(1 == wCfgLoad)
	{
		memset(&cfg_cpy, 0, sizeof(cfg_cpy));
		strcpy(cfg_cpy.modname, "cfg_dat");
		cfg_cpy.error = var_rd(&cfg_cpy);

		if (cfg_cpy.error!=0)
		{
  			DMSTATUS = cfg_cpy.error;
  		}
		else
		{
			wCfgLoad = 0;
  		}
	}
}  /* end of _CYCLIC */

/********************************************************************
                                                          Function
********************************************************************/
unsigned short	var_rd(var_rd_typ	*var_rd_ptr)
{

	/* Internal PV */
	float  					 value=0;
	long			    	longvalue=0;
	unsigned  long  		DA_ID;
	plcbit 			  	*bitval;                 /*    !                     */
	unsigned  char 	   *bval;                   /*    !                     */
	float 					 *fval;                   /*    !                     */
	short 					*i16val;                 /*    !                     */
	long 					*i32val;                 /*    !                     */
	char 					*i8val;                  /*    !                     */
	unsigned  long 		*lval;                    /*    !                     */
	unsigned short 		*wval;                   /*    !                     */
	char					*var_start_ptr,*full_line_ptr;
	char					*var_end_ptr;
	char					*val_start_ptr;
	char				 	*val_end_ptr;
	unsigned  long  		pv_adr;
	unsigned  long  		pv_len;
	char					    IPtyp;
	unsigned  long  	   dat_adr;
	unsigned short  	   dimension;
	long  					    PV_adr;
	char		  			  *PV_ptr;

	unsigned  long  		line_adr;
	unsigned short  		status;
	unsigned  long  		type;

	long				        end_adr,line_start_adr;
	char					* line_start_ptr;
	unsigned  long  	   length;                 /*    !                     */

	DatObjInfo_typ		   fDOInfo;

	/****************************************************************************************/
	/* Get PV initialization DM information */
	fDOInfo.enable    = 1;
	fDOInfo.pName     = (UDINT)var_rd_ptr->modname;
	DatObjInfo(&fDOInfo);
	DA_ID   = fDOInfo.ident;
	dat_adr = fDOInfo.pDatObjMem;
	length  = fDOInfo.len;
	IPtyp   = fDOInfo.MemType;
	status  = fDOInfo.status;
	if (status != 0)
	{
		strcpy(DM_ER_STR, "DatObjInfo: DM read error");
		return status;
	}
	/* Allocate memory for PV lines */
	status = TMP_alloc(100, (void*)&(line_adr));
	if (status != 0)
	{
		strcpy(DM_ER_STR, "TMP_alloc: lines memory allocate error");
		return status;
	}
	line_start_ptr 	= (char*)dat_adr;
	full_line_ptr 	= (char*)line_adr;
	/* Allocate memory for PV */
	status = TMP_alloc(100,(void*)&(PV_adr));
	if (status != 0)
	{
		strcpy(DM_ER_STR, "TMP_alloc: PV memory allocate error");
		return status;
	}
	PV_ptr = (char*)PV_adr;
	var_rd_ptr->line_no = 0;
	end_adr = dat_adr+length-3;
	line_start_adr = (long)(line_start_ptr);
	while (line_start_adr < end_adr)  /*****while (*line_start_ptr != 'e')           */
	{
		var_rd_ptr->line_no++;
		strncpy(full_line_ptr,line_start_ptr,100);
		var_start_ptr =full_line_ptr;
		while ((*var_start_ptr ==' ')||(*var_start_ptr =='"'))		/* Suche Variable Start */
		{
			var_start_ptr++;
		}
		var_end_ptr = var_start_ptr;		/* Suche Variable Ende  */
		while ((*var_end_ptr !=' ') && (*var_end_ptr !='='))
		{
			var_end_ptr++;
		}
		val_start_ptr = var_end_ptr;
		while ((*val_start_ptr ==' ') || (*val_start_ptr =='='))
		{
			val_start_ptr++;
		}
		val_end_ptr = val_start_ptr;
		while ((*val_end_ptr !=' ') && (*val_end_ptr !=0))		/* Suche Variable Start */
		{
			val_end_ptr++;
		}
		*var_end_ptr = 0;		/* Nullterminierung */
		*val_end_ptr = 0;		/* Nullterminierung */
		strcpy(PV_ptr,var_rd_ptr->taskname);	/* Zusammensetzung der Variable */
		if (strlen(var_rd_ptr->taskname)!=0)
		{
			strcat(PV_ptr, ":");
		} /*if*/
		if (strlen(var_rd_ptr->pre_string)!=0)
		{
			strcat(PV_ptr, var_rd_ptr->pre_string);
		}
		strcat(PV_ptr, var_start_ptr);
		/* Get PV address */
		status = PV_xgetadr((char*)PV_ptr, &(pv_adr), &(pv_len)) ;
		if (status != 0)
		{
			strcpy(DM_ER_STR, "PV_xgetadr: PV address get error");
			return status;
		}
		/* Get PV information */
		status = PV_ninfo((char*)PV_ptr, &(type), &(pv_len), &(dimension)) ;
		if (status != 0)
		{
			strcpy(DM_ER_STR, "PV_ninfo: PV information get error");
			return status;
		}
		line_start_ptr += strlen(line_start_ptr);
		line_start_ptr++;
		line_start_adr = (long)line_start_ptr;
		if (type == 8) /**** FLOAT )*/
		{
			value =	atof((unsigned long) (val_start_ptr));
		}
		else
		{
			longvalue = atoi((unsigned long) (val_start_ptr)); /* strtol(val_start_ptr, 0, 0); */
		}
		switch ((unsigned short)(type))
		{
			case 1: /**** BIT                                                 */
				bitval  = (plcbit *)pv_adr ;
				*bitval = (unsigned)((long)(longvalue)) ;
				break;
			case 2: /**** INT8                                                */
				i8val  = (char *)pv_adr ;
				*i8val = (char)((long)(longvalue)) ;
				break;
			case 3: /**** INT16                                               */
				i16val  = (short *)pv_adr;
				*i16val = (short)((long)(longvalue));
				break;
			case 4: /**** INT32                                               */
				i32val  = (long *)pv_adr;
				*i32val = (long)(longvalue);
				break;
			case 5: /**** BYTE                                                */
				bval  = (unsigned char *)pv_adr;
				*bval = (unsigned char)((unsigned long)(longvalue));
				break;
			case 6: /**** WORD                                                */
				wval  = (unsigned short *)pv_adr ;
				*wval = (unsigned short)((unsigned long)(longvalue));
				break;
			case 7: /**** LONG                                                */
				lval  = (unsigned long *)pv_adr ;
				*lval = (unsigned long)(longvalue);
				break;
			case 8: /**** FLOAT                                               */
				fval  = (float *)pv_adr;
				*fval = value;
				break;
			default:
				break;
		} /* End of switch */
	} /* End of while (line_start_adr < end_adr) */
	/* Free memory for PV */
	status = TMP_free(100, (void*)PV_ptr);
	if (status != 0)
	{
		strcpy(DM_ER_STR, "TMP_free: PV memory free error");
		return status;
	}
	/* Free memory for PV lines */
	status = TMP_free(100, (void*)line_adr);
	if (status != 0)
	{
		strcpy(DM_ER_STR, "TMP_free: line memory free error");
		return status;
	}

	return status;
} /* End of var_rd function */
```

#### cfg_cpy.var - Local variables
```iecst
VAR
	wCfgLoad : USINT;
	cfg_cpy : var_rd_typ;
	DMSTATUS : INT;
	DM_ER_STR : STRING[48];
END_VAR
```

### Data object Logical/recipeMan/var_fix (Simple, version 1.00.0) - Variable once save / load

#### var_fix.dat
```
;********************************************************************************************
;var,array or struct configuration!
;********************************************************************************************
;fill the blank up to 31 chars and cann't use'tab' key
;maxmim 50 lines
;"                               "
;***************************************
"gT_Par.Fix                     " ;1
"gAccuLinear                    " ;2
"gServoLinear                   " ;3
"gHeatingPlan                   " ;4
"gThickProf.FunOption           " ;5
"gThickProf.ShareSet            " ;6
"LMold.ValveDelay               " ;7
"RMold.ValveDelay               " ;8
"gMachineFix                    " ;9
"gSPC_Par                       " ;10
;***************************************
"gThickFix                      " ;11
"gUserFix                       " ;12
"gUserFix_new                   " ;13
"                               " ;14
"                               " ;15
"                               " ;16
"                               " ;17
"                               " ;18
"                               " ;19
"                               " ;20
;***************************************
"                               " ;21
"                               " ;22
"                               " ;23
"                               " ;24
"                               " ;25
"                               " ;26
"                               " ;27
"                               " ;28
"                               " ;29
"                               " ;30
;***************************************
"                               " ;31
"                               " ;32
"                               " ;33
"                               " ;34
"                               " ;35
"                               " ;36
"                               " ;37
"                               " ;38
"                               " ;39
"                               " ;40
;***************************************
"                               " ;41
"                               " ;42
"                               " ;43
"                               " ;44
"                               " ;45
"                               " ;46
"                               " ;47
"                               " ;48
"                               " ;49
"                               " ;50
;*************************************** end
```

### Data object Logical/recipeMan/var_mold (Simple, version 1.00.0) - Variable multiple save /load

#### var_mold.dat
```
;********************************************************************************************
;var,array or struct configuration!
;********************************************************************************************
;fill the blank up to 31 chars and cann't use'tab' key
;maxmim 50 lines
;"                               "
"gT_Par.Par                     " ;1
"gMachinePara                   " ;2
"LMold.TimeSet                  " ;3
"RMold.TimeSet                  " ;4
"gMacOption                     " ;5
"gThickProf.TimSet              " ;6
"gThickProf.AccuSet             " ;7
"usScaleIndex                   " ;8
"gUserPara                      " ;9
"                               " ;10
;***************************************
"                               " ;11
"                               " ;12
"                               " ;13
"                               " ;14
"                               " ;15
"                               " ;16
"                               " ;17
"                               " ;18
"                               " ;19
"                               " ;20
;***************************************
"                               " ;21
"                               " ;22
"                               " ;23
"                               " ;24
"                               " ;25
"                               " ;26
"                               " ;27
"                               " ;28
"                               " ;29
"                               " ;30
;***************************************
"                               " ;31
"                               " ;32
"                               " ;33
"                               " ;34
"                               " ;35
"                               " ;36
"                               " ;37
"                               " ;38
"                               " ;39
"                               " ;40
;***************************************
"                               " ;41
"                               " ;42
"                               " ;43
"                               " ;44
"                               " ;45
"                               " ;46
"                               " ;47
"                               " ;48
"                               " ;49
"                               " ;50
;*************************************** end
```

### Data object Logical/recipeMan/cfg_dat (Simple, version 1.00.0) - Config temperature data

#### cfg_dat.dat
```
;********************************************************************************************
;                                                Project parameters configuration!
;********************************************************************************************

;TEMPERATURE - 00;
"gT_Par.Fix.Enable[0]            = 1     "
"gT_Par.Fix.Enable[1]            = 1     "
"gT_Par.Fix.Enable[2]            = 1     "
"gT_Par.Fix.Enable[3]            = 1     "
"gT_Par.Fix.Enable[4]            = 1     "
"gT_Par.Fix.Enable[5]            = 1     "
"gT_Par.Fix.Enable[6]            = 1     "
"gT_Par.Fix.Enable[7]            = 1     "
"gT_Par.Fix.Enable[8]            = 1     "
"gT_Par.Fix.Enable[9]            = 1     "
"gT_Par.Fix.Enable[10]           = 1     "
"gT_Par.Fix.Enable[11]           = 1     "
"gT_Par.Fix.Enable[12]           = 1     "
"gT_Par.Fix.Enable[13]           = 1     "
"gT_Par.Fix.Enable[14]           = 1     "
"gT_Par.Fix.Enable[15]           = 1     "
"gT_Par.Fix.Enable[16]           = 1     "
```

### Package Logical/Heating - zone heating and cooling

### Program Logical/Heating/h_pid (ANSIC, version 1.00.0) - heating PID
